{attribute 'hide'}
INTERFACE INTERNAL StringBuilder

METHOD Append : StringBuilder // Append text TO t current build STRING.
VAR_INPUT
    Text : Tc2_System.T_MaxString; //Text to append to current build string
END_VAR
END_METHOD

METHOD AppendIf : StringBuilder
VAR_INPUT
    Condition : BOOL;
    Text : Tc2_System.T_MaxString;
END_VAR
END_METHOD

METHOD InsertAtLocation : StringBuilder
VAR_INPUT
    Text : Tc2_System.T_MaxString;
    Position : INT;
END_VAR
END_METHOD

METHOD PadLeft : StringBuilder
VAR_INPUT
    text : Tc2_System.T_MaxString; // Text to append to current build string
    length : INT; // Total length of text + padding
    c : STRING(1); // Character to be padded left of text
END_VAR
END_METHOD

METHOD Reset : LimitedStringBuilder //Reset current build STRING TO an empty STRING.
END_METHOD

METHOD ToString : Tc2_System.T_MaxString //Returns current build STRING.
END_METHOD

END_INTERFACE

(* stored: Version 1.1.0.1
   Itf StringBuilder: Id {6e140e27-b917-4c21-b37e-0ed41ff5a291}
   Method Append: Id {258ee2c9-d57d-4edd-a271-999221890c73}
   Method AppendIf: Id {c52057ff-21ee-443b-a5ea-eec9f48e03c8}
   Method InsertAtLocation: Id {f2e89a85-4a3f-4b63-9268-57936f9e9b1a}
   Method PadLeft: Id {08ee748e-fc3a-42c5-a97c-478fc4802754}
   Method Reset: Id {25884b9e-bd34-45c8-b59c-5eaa0d8be981}
   Method ToString: Id {63021287-748e-49ec-b934-c7db98fd5041} *)
